Universal Robots PolyScope program: rtde_control_loop_kendama.urp

Program rtde_control_loop_kendama (installation=default directory=/programs/usbdisk/universal createdIn=3.2.19275.0 lastSavedIn=5.9.5.1031259 robotSerialNumber=20195500451)
Calibrated DH parameters: a=[0.00002, -0.231658, -0.317125, 0.000011, 0.000055, 0]; d=[0.162082, 123.190176, -180.284242, 57.22734, 0.099524, 0.09934]; alpha=[1.569304, 0.00289, 0.004025, 1.569925, -1.569026, 0]; deltaTheta=[0, 0.993923, 4.662183, 0.627072, 0.000001, 0]
BeforeStart
  ctrl_type := 0
  selection_vec := [0,0,0,0,0,0]
  wrench := [0,0,0,0,0,0]
  limits := [0,0,0,0,0,0]
  tmp := [0,0,0,0,0,0,0,0,0,0,0,0,0,0,0,0,0,0,0]
  Script: rtde_set_watchdog("input_int_register_0", 0.5, "STOP")
  Script: zero_ftsensor()
Robot Program (runOnlyOnce=false)
  If ctrl_type == 1
    Script: servoj([tmp[1],tmp[2],tmp[3],tmp[4],tmp[5],tmp[6]],tmp[7],tmp[8],tmp[9],tmp[10],tmp[11])
  ElseIf ctrl_type == 2
    SuppressedNode
      Script: speedj([tmp[1],tmp[2],tmp[3],tmp[4],tmp[5],tmp[6]],tmp[7],tmp[8])
    If tmp[8]==0
      Script: speedj([tmp[1],tmp[2],tmp[3],tmp[4],tmp[5],tmp[6]],tmp[7])
    Else 
      Script: speedj([tmp[1],tmp[2],tmp[3],tmp[4],tmp[5],tmp[6]],tmp[7],tmp[8])
  ElseIf ctrl_type == 3
    Script: movej([tmp[1],tmp[2],tmp[3],tmp[4],tmp[5],tmp[6]],tmp[7],tmp[8],tmp[9],tmp[10])
  ElseIf ctrl_type == 4
    Script: movel(p[tmp[1],tmp[2],tmp[3],tmp[4],tmp[5],tmp[6]],tmp[7],tmp[8],tmp[9],tmp[10])
  ElseIf ctrl_type == 5
    Script: speedl([tmp[1],tmp[2],tmp[3],tmp[4],tmp[5],tmp[6]],tmp[7],tmp[8],tmp[9])
    If tmp[8]==0
      Script: speedl([tmp[1],tmp[2],tmp[3],tmp[4],tmp[5],tmp[6]],tmp[7],aRot=tmp[9])
    Else 
      Script: speedl([tmp[1],tmp[2],tmp[3],tmp[4],tmp[5],tmp[6]],tmp[7],tmp[8],tmp[9])
  ElseIf ctrl_type == 6
    Script: force_mode(Base,selection_vec,wrench,2,limits)
  ElseIf ctrl_type == 7
    Script: stopj(tmp[1])
  ElseIf ctrl_type == 8
    q_from_ik := get_inverse_kin(p[tmp[1],tmp[2],tmp[3],tmp[4],tmp[5],tmp[6]],[tmp[7],tmp[8],tmp[9],tmp[10],tmp[11],tmp[12]],0.0001,0.001)
    If q_from_ik[1]≥.04
      Script: stopj(2)
    Else 
      SuppressedNode
        Loop While (checkContinuously=false) expression=norm(q-q_from_ik)>1
          SuppressedNode
            q_from_ik := get_inverse_kin(p[tmp[1],tmp[2],tmp[3],tmp[4],tmp[5],tmp[6]],[tmp[7],tmp[8],tmp[9],tmp[10],tmp[11],tmp[12]],0.0001,0.001)
      qnorm := norm(q-q_from_ik)
      Loop While (checkContinuously=false) expression=qnorm>1
        q_from_ik := get_inverse_kin(p[tmp[1],tmp[2],tmp[3],tmp[4],tmp[5],tmp[6]],[tmp[7],tmp[8],tmp[9],tmp[10],tmp[11],tmp[12]],0.0001,0.001)
        qnorm := norm(q-q_from_ik)
      Script: servoj(q_from_ik,tmp[13],tmp[14],tmp[15],tmp[16],tmp[17])
  SuppressedNode
    Script: sync()
  args := [tmp[7],tmp[8],tmp[9],tmp[10],tmp[1]]
Thread Thread_1 (runOnlyOnce=false)
  Folder Read remote registers
    tmp := [0,0,0,0,0,0,0,0,0,0,0,0,0,0,0,0,0,0,0]
    Script: tmp[0] = read_input_float_register(0)
    Script: tmp[1] = read_input_float_register(1)
    Script: tmp[2] = read_input_float_register(2)
    Script: tmp[3] = read_input_float_register(3)
    Script: tmp[4] = read_input_float_register(4)
    Script: tmp[5] = read_input_float_register(5)
    Script: tmp[6] = read_input_float_register(6)
    Script: tmp[7] = read_input_float_register(7)
    Script: tmp[8] = read_input_float_register(8)
    Script: tmp[9] = read_input_float_register(9)
    Script: tmp[10] = read_input_float_register(10)
    Script: tmp[11] = read_input_float_register(11)
    Script: tmp[12] = read_input_float_register(12)
    Script: tmp[13] = read_input_float_register(13)
    Script: tmp[14] = read_input_float_register(14)
    Script: tmp[15] = read_input_float_register(15)
    Script: tmp[16] = read_input_float_register(16)
    Script: tmp[17] = read_input_float_register(17)
    Script: tmp[18] = read_input_float_register(18)
    ctrl_type := tmp[0]
    If ctrl_type ==6
      wrench := [tmp[1],tmp[2],tmp[3],tmp[4],tmp[5],tmp[6]]
      selection_vec := [tmp[7],tmp[8],tmp[9],tmp[10],tmp[11],tmp[12]]
      limits := [tmp[13],tmp[14],tmp[15],tmp[16],tmp[17],tmp[18]]
  Script: sync()
Thread Thread_2 (runOnlyOnce=false)
  Folder Send Torque Values
    torque := get_joint_torques()
    Script: write_output_float_register(0, torque[0])
    Script: write_output_float_register(1, torque[1])
    Script: write_output_float_register(2, torque[2])
    Script: write_output_float_register(3, torque[3])
    Script: write_output_float_register(4, torque[4])
    Script: write_output_float_register(5, torque[5])
    Script: write_output_boolean_register(64, is_steady())
    q := get_actual_joint_positions()
    tcp := get_actual_tcp_pose()
    Script: sync()
